_CFC_ (* Continuous Function Chart, elements in execution order *)
#0 FT_Ostanov:F_TRIG(CLK: SHU6_PV1_UST_RE_OSTANOV)
#1 TOF_Progrev:TOF(IN: SHU6_PV1_UST_RE_PROGREV, PT: T#1s)
#2 AND(#1.Q, SHU6_PV1_UST_SOST_OTKL)
#3 OR(#0.Q, SHU6_PV1_Z_POZH, SHU6_PV1_Z_NET_VH_NAPR, SHU6_PV1_Z_OTKAZ_VTORICH_SEP, SHU6_PV1_Z_GVS1_OTKAZ, #2, Z_ZAM_SR, SHU6_PV1_Z_YA2_OTKAZ, SHU6_PV1_HZ20S60, MP1_OTKAZ)
#4 SHU6_PV1_UST_SET_STOP <= #3
#5 sr_stop:SR(SET1: #3, RESET: SHU6_PV1_UST_SOST_VKL)
#6 SHU6_PV1_UST_RE_STOP <= #5.Q1
_END_CFC_
(* the same logic as Structured Text *)
FT_Ostanov(CLK := SHU6_PV1_UST_RE_OSTANOV);
TOF_Progrev(IN := SHU6_PV1_UST_RE_PROGREV, PT := T#1s);
_t19 := FT_Ostanov.Q OR SHU6_PV1_Z_POZH OR SHU6_PV1_Z_NET_VH_NAPR OR SHU6_PV1_Z_OTKAZ_VTORICH_SEP OR SHU6_PV1_Z_GVS1_OTKAZ OR (TOF_Progrev.Q AND SHU6_PV1_UST_SOST_OTKL) OR Z_ZAM_SR OR SHU6_PV1_Z_YA2_OTKAZ OR SHU6_PV1_HZ20S60 OR MP1_OTKAZ;
SHU6_PV1_UST_SET_STOP := _t19;
sr_stop(SET1 := _t19, RESET := SHU6_PV1_UST_SOST_VKL);
SHU6_PV1_UST_RE_STOP := sr_stop.Q1;
END_PROGRAM

(* POU Regim/Ostanov, CFC *)
PROGRAM Ostanov
VAR
	RT_OTKL: R_TRIG;
	SR_OSTANOV: SR;
	TON_AVR_M: TON;
	Z_zam_ostatov: R_TRIG;
END_VAR
VAR (* helpers for the ST form of the networks *)
	_t31 : BOOL;
END_VAR
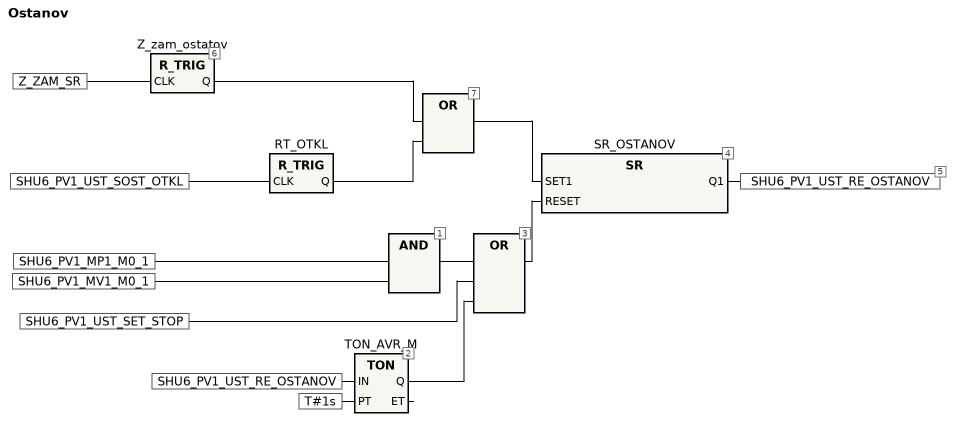
_CFC_ (* Continuous Function Chart, elements in execution order *)
#0 RT_OTKL:R_TRIG(CLK: SHU6_PV1_UST_SOST_OTKL)
#1 AND(SHU6_PV1_MP1_M0_1, SHU6_PV1_MV1_M0_1)
#2 TON_AVR_M:TON(IN: SHU6_PV1_UST_RE_OSTANOV, PT: T#1s)
#3 OR(#1, SHU6_PV1_UST_SET_STOP, #2.Q)
#4 SR_OSTANOV:SR(SET1: #7, RESET: #3)
#5 SHU6_PV1_UST_RE_OSTANOV <= #4.Q1
#6 Z_zam_ostatov:R_TRIG(CLK: Z_ZAM_SR)
#7 OR(#6.Q, #0.Q)
_END_CFC_
(* the same logic as Structured Text *)
RT_OTKL(CLK := SHU6_PV1_UST_SOST_OTKL);
TON_AVR_M(IN := SHU6_PV1_UST_RE_OSTANOV, PT := T#1s);
SR_OSTANOV(SET1 := _t31, RESET := (SHU6_PV1_MP1_M0_1 AND SHU6_PV1_MV1_M0_1) OR SHU6_PV1_UST_SET_STOP OR TON_AVR_M.Q);
SHU6_PV1_UST_RE_OSTANOV := SR_OSTANOV.Q1;
Z_zam_ostatov(CLK := Z_ZAM_SR);
_t31 := Z_zam_ostatov.Q OR RT_OTKL.Q;
END_PROGRAM

(* POU Regim/Progrev, CFC *)
PROGRAM Progrev
VAR
	RS_Progrev: RS;
	RT_VKL: R_TRIG;
	TON_SHU6_PV1_TE6_M_UST: TON;
	SR_First_On: SR;
END_VAR
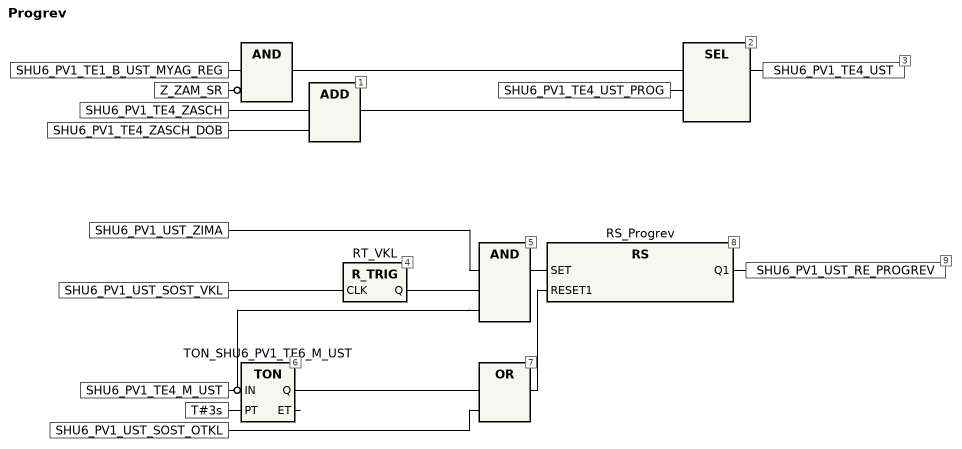
_CFC_ (* Continuous Function Chart, elements in execution order *)
#0 AND(SHU6_PV1_TE1_B_UST_MYAG_REG, NOT Z_ZAM_SR)
#1 ADD(SHU6_PV1_TE4_ZASCH, SHU6_PV1_TE4_ZASCH_DOB)
#2 SEL(#0, SHU6_PV1_TE4_UST_PROG, #1)
#3 SHU6_PV1_TE4_UST <= #2
#4 RT_VKL:R_TRIG(CLK: SHU6_PV1_UST_SOST_VKL)
#5 AND(SHU6_PV1_UST_ZIMA, #4.Q, SHU6_PV1_TE4_M_UST)
#6 TON_SHU6_PV1_TE6_M_UST:TON(IN: NOT SHU6_PV1_TE4_M_UST, PT: T#3s)
#7 OR(#6.Q, SHU6_PV1_UST_SOST_OTKL)
#8 RS_Progrev:RS(SET: #5, RESET1: #7)
#9 SHU6_PV1_UST_RE_PROGREV <= #8.Q1
_END_CFC_
(* the same logic as Structured Text *)
SHU6_PV1_TE4_UST := SEL(SHU6_PV1_TE1_B_UST_MYAG_REG AND NOT Z_ZAM_SR, SHU6_PV1_TE4_UST_PROG, SHU6_PV1_TE4_ZASCH + SHU6_PV1_TE4_ZASCH_DOB);
RT_VKL(CLK := SHU6_PV1_UST_SOST_VKL);
TON_SHU6_PV1_TE6_M_UST(IN := NOT SHU6_PV1_TE4_M_UST, PT := T#3s);
RS_Progrev(SET := SHU6_PV1_UST_ZIMA AND RT_VKL.Q AND SHU6_PV1_TE4_M_UST, RESET1 := TON_SHU6_PV1_TE6_M_UST.Q OR SHU6_PV1_UST_SOST_OTKL);
SHU6_PV1_UST_RE_PROGREV := RS_Progrev.Q1;
END_PROGRAM

(* POU Regim/Pusk, CFC *)
PROGRAM Pusk
VAR
	RS_Pusk: RS;
	FT_PROGREV: F_TRIG;
	RT_VKL: R_TRIG;
	TON_sost_VKL: TON;
	TON_AVR_M: TON;
	re_start: F_TRIG;
	TON_Z_ZAM: TON;
END_VAR
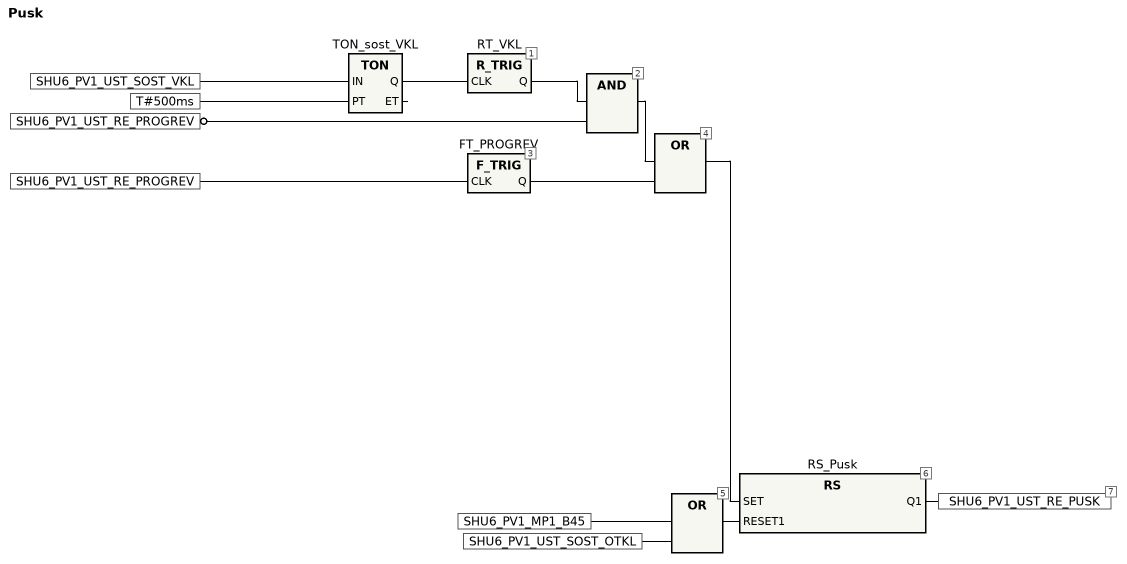
_CFC_ (* Continuous Function Chart, elements in execution order *)
#0 TON_sost_VKL:TON(IN: SHU6_PV1_UST_SOST_VKL, PT: T#500ms)
#1 RT_VKL:R_TRIG(CLK: #0.Q)
#2 AND(#1.Q, NOT SHU6_PV1_UST_RE_PROGREV)
#3 FT_PROGREV:F_TRIG(CLK: SHU6_PV1_UST_RE_PROGREV)
#4 OR(#2, #3.Q)
#5 OR(SHU6_PV1_MP1_B45, SHU6_PV1_UST_SOST_OTKL)
#6 RS_Pusk:RS(SET: #4, RESET1: #5)
#7 SHU6_PV1_UST_RE_PUSK <= #6.Q1
_END_CFC_
(* the same logic as Structured Text *)
TON_sost_VKL(IN := SHU6_PV1_UST_SOST_VKL, PT := T#500ms);
RT_VKL(CLK := TON_sost_VKL.Q);
FT_PROGREV(CLK := SHU6_PV1_UST_RE_PROGREV);
RS_Pusk(SET := (RT_VKL.Q AND NOT SHU6_PV1_UST_RE_PROGREV) OR FT_PROGREV.Q, RESET1 := SHU6_PV1_MP1_B45 OR SHU6_PV1_UST_SOST_OTKL);
SHU6_PV1_UST_RE_PUSK := RS_Pusk.Q1;
END_PROGRAM

(* POU Regim/Rabota, CFC *)
PROGRAM Rabota
VAR
	RS_Rabota: RS;
	FT_Pusk: F_TRIG;
END_VAR
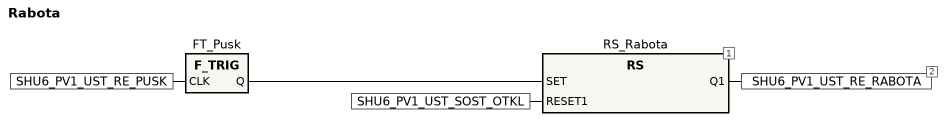
_CFC_ (* Continuous Function Chart, elements in execution order *)
#0 FT_Pusk:F_TRIG(CLK: SHU6_PV1_UST_RE_PUSK)
#1 RS_Rabota:RS(SET: #0.Q, RESET1: SHU6_PV1_UST_SOST_OTKL)
#2 SHU6_PV1_UST_RE_RABOTA <= #1.Q1
_END_CFC_
(* the same logic as Structured Text *)
FT_Pusk(CLK := SHU6_PV1_UST_RE_PUSK);
RS_Rabota(SET := FT_Pusk.Q, RESET1 := SHU6_PV1_UST_SOST_OTKL);
SHU6_PV1_UST_RE_RABOTA := RS_Rabota.Q1;
END_PROGRAM

(* POU IM/ALL_IM, CFC *)
PROGRAM ALL_IM
VAR
END_VAR
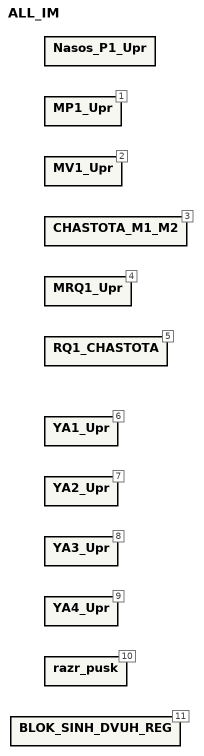
_CFC_ (* Continuous Function Chart, elements in execution order *)
#0 Nasos_P1_Upr()
#1 MP1_Upr()
#2 MV1_Upr()
#3 CHASTOTA_M1_M2()
#4 MRQ1_Upr()
#5 RQ1_CHASTOTA()
#6 YA1_Upr()
#7 YA2_Upr()
#8 YA3_Upr()
#9 YA4_Upr()
#10 razr_pusk()
#11 BLOK_SINH_DVUH_REG()
_END_CFC_
(* the same logic as Structured Text *)
Nasos_P1_Upr();
MP1_Upr();
MV1_Upr();
CHASTOTA_M1_M2();
MRQ1_Upr();
RQ1_CHASTOTA();
YA1_Upr();
YA2_Upr();
YA3_Upr();
YA4_Upr();
razr_pusk();
BLOK_SINH_DVUH_REG();
END_PROGRAM

(* POU IM/Nasos_P1_Upr, CFC *)
PROGRAM Nasos_P1_Upr
VAR
	fb_HVACMS_P1: FB_HVACMotor1Speed;
	SR_P1: SR;
	startDelay_P1: TIME := T#0s;
	stopDelay_P1: TIME := T#0s;
	delayFBC_P1: TIME:=T#5s ;
	feedbPT_P1: TIME :=T#10s ;
	delayFBP_P1: TIME := T#10s;
	TON_P1_OTKL_Leto: TON;
	TON_P1_VKL_Leto: TON;
END_VAR
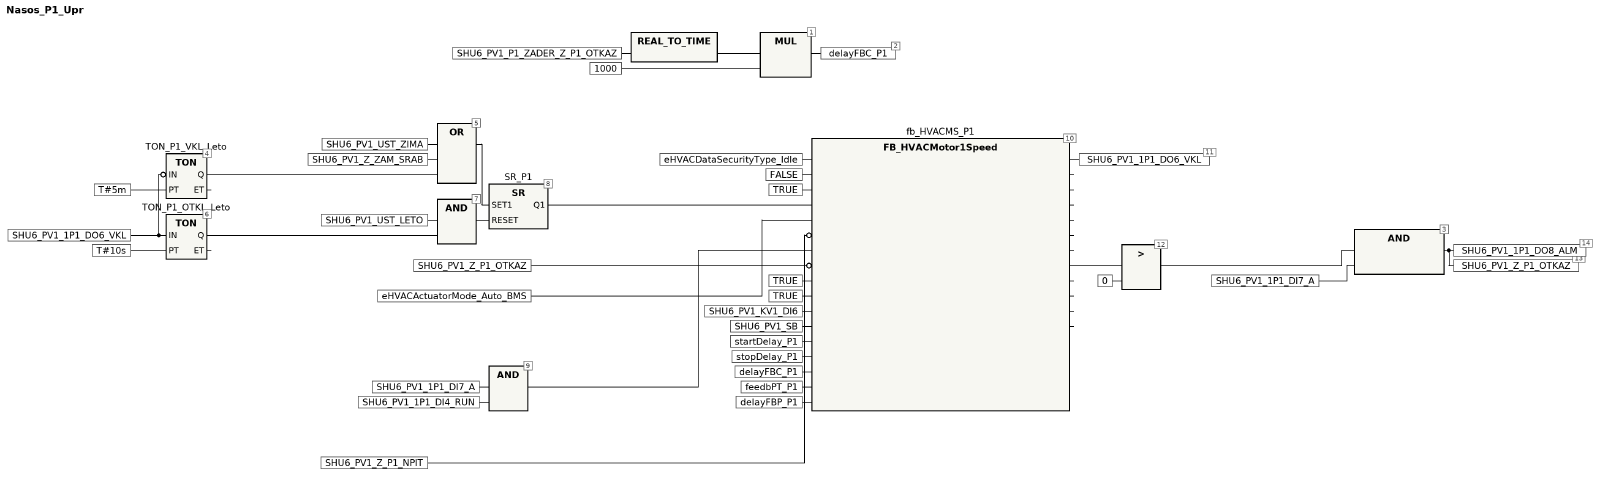
